Omron CX-Programmer project NuevoProyecto (CX-Programmer 9.61)

# PLC Practica2E1: CJ2M CPU11

## Global symbols (name address type ; comment)
1.03 BOOL  ; 1.03
T0 CHANNEL  ; #30

## Program NuevoPrograma1 (cyclic task 0)
Local symbols
Amarillo1 1.01 BOOL  ; 1.01
Amarillo2 1.09 BOOL  ; 1.09
Ciclo1min 1.03 BOOL  ; 1.03
Entrada1 0.00 BOOL  ; 0.00
Entrada15 0.15 BOOL  ; 0.15
Entrada2 0.01 BOOL  ; 0.01
Rojo1 1.00 BOOL  ; 1.00
Rojo2 1.08 BOOL  ; 1.08
Verde1 1.02 BOOL  ; 1.02
Verde2 1.10 BOOL  ; 1.10

### Section Sección1

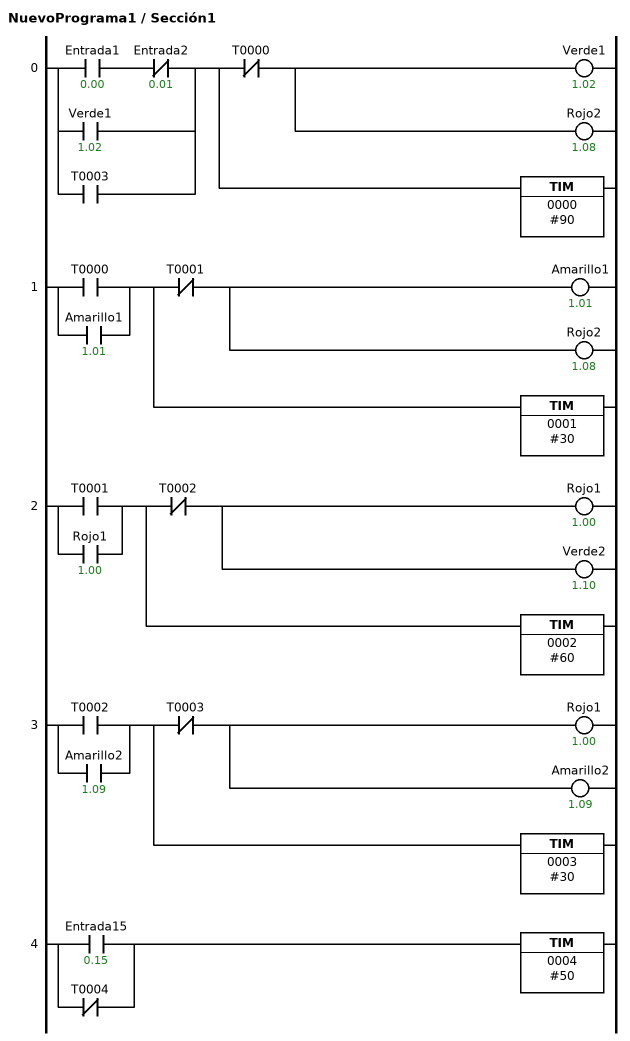
; rung 0
LD Entrada1  ; 0.00
ANDNOT Entrada2  ; 0.01
OR Verde1  ; 1.02
OR T0003
OUT TR0
ANDNOT T0000
OUT Verde1  ; 1.02
OUT Rojo2  ; 1.08
LD TR0
TIM 0000 #90
; rung 1
LD T0000
OR Amarillo1  ; 1.01
OUT TR0
ANDNOT T0001
OUT Amarillo1  ; 1.01
OUT Rojo2  ; 1.08
LD TR0
TIM 0001 #30
; rung 2
LD T0001
OR Rojo1  ; 1.00
OUT TR0
ANDNOT T0002
OUT Rojo1  ; 1.00
OUT Verde2  ; 1.10
LD TR0
TIM 0002 #60
; rung 3
LD T0002
OR Amarillo2  ; 1.09
OUT TR0
ANDNOT T0003
OUT Rojo1  ; 1.00
OUT Amarillo2  ; 1.09
LD TR0
TIM 0003 #30
; rung 4
LD Entrada15  ; 0.15
ORNOT T0004
TIM 0004 #50

### Section END
; rung 0
END(001)